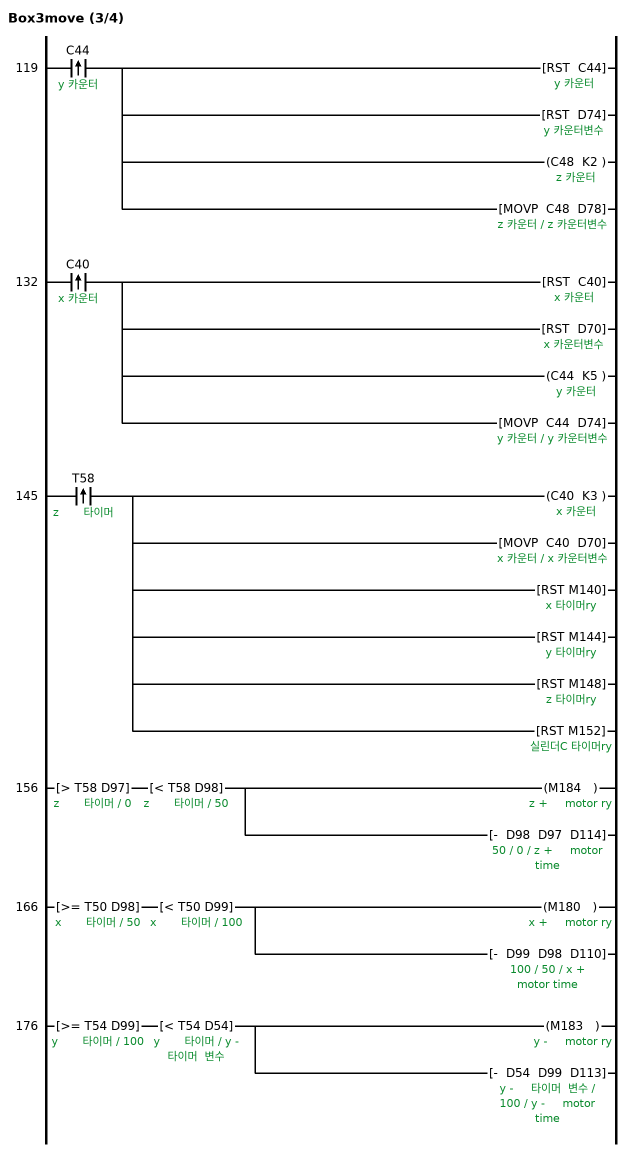
[picture p24: ladder of Box3move, rungs at steps 119 to 176]
119   LDP     C44  ; y 카운터
      RST     C44  ; y 카운터
      RST     D74  ; y 카운터변수
      OUT     C48 K2  ; z 카운터
      MOVP    C48 D78
132   LDP     C40  ; x 카운터
      RST     C40  ; x 카운터
      RST     D70  ; x 카운터변수
      OUT     C44 K5  ; y 카운터
      MOVP    C44 D74
145   LDP     T58  ; z       타이머
      OUT     C40 K3  ; x 카운터
      MOVP    C40 D70
      RST     M140  ; x 타이머ry
      RST     M144  ; y 타이머ry
      RST     M148  ; z 타이머ry
      RST     M152  ; 실린더C 타이머ry
156   LD>     T58 D97  ; z       타이머 / 0
      AND<    T58 D98  ; z       타이머 / 50
      OUT     M184  ; z +     motor ry
      -       D98 D97 D114  ; z +     motor time
166   LD>=    T50 D98  ; x       타이머 / 50
      AND<    T50 D99  ; x       타이머 / 100
      OUT     M180  ; x +     motor ry
      -       D99 D98 D110  ; x +     motor time
176   LD>=    T54 D99  ; y       타이머 / 100
      AND<    T54 D54  ; y       타이머 / y -     타이머  변수
      OUT     M183  ; y -     motor ry
      -       D54 D99 D113  ; y -     motor time
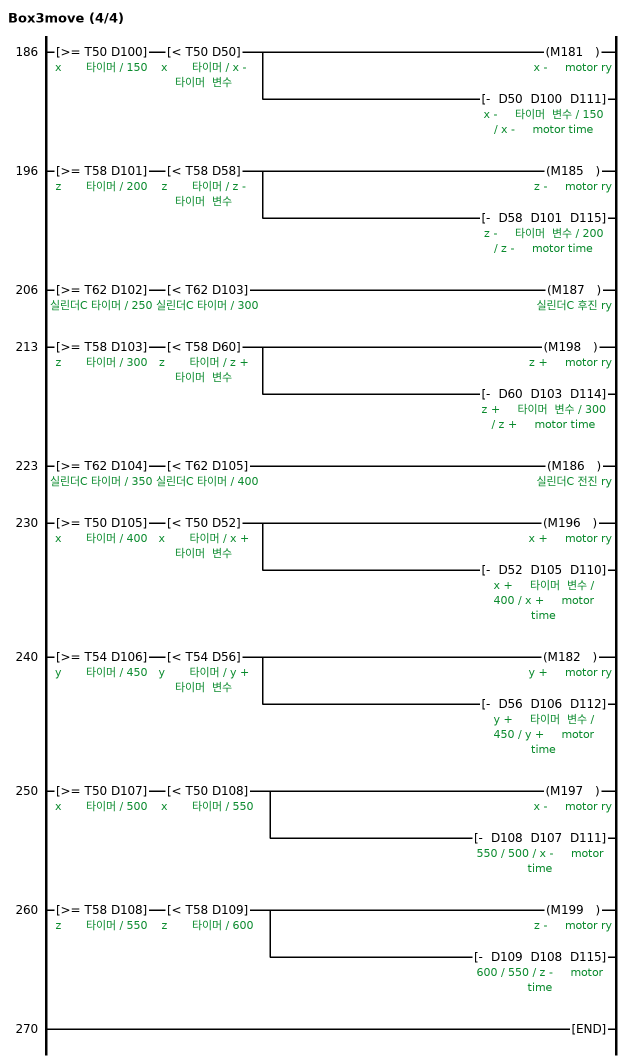
186   LD>=    T50 D100  ; x       타이머 / 150
      AND<    T50 D50  ; x       타이머 / x -     타이머  변수
      OUT     M181  ; x -     motor ry
      -       D50 D100 D111  ; x -     motor time
196   LD>=    T58 D101  ; z       타이머 / 200
      AND<    T58 D58  ; z       타이머 / z -     타이머  변수
      OUT     M185  ; z -     motor ry
      -       D58 D101 D115  ; z -     motor time
206   LD>=    T62 D102  ; 실린더C 타이머 / 250
      AND<    T62 D103  ; 실린더C 타이머 / 300
      OUT     M187  ; 실린더C 후진 ry
213   LD>=    T58 D103  ; z       타이머 / 300
      AND<    T58 D60  ; z       타이머 / z +     타이머  변수
      OUT     M198  ; z +     motor ry
      -       D60 D103 D114
223   LD>=    T62 D104  ; 실린더C 타이머 / 350
      AND<    T62 D105  ; 실린더C 타이머 / 400
      OUT     M186  ; 실린더C 전진 ry
230   LD>=    T50 D105  ; x       타이머 / 400
      AND<    T50 D52  ; x       타이머 / x +     타이머  변수
      OUT     M196  ; x +     motor ry
      -       D52 D105 D110
240   LD>=    T54 D106  ; y       타이머 / 450
      AND<    T54 D56  ; y       타이머 / y +     타이머  변수
      OUT     M182  ; y +     motor ry
      -       D56 D106 D112  ; y +     motor time
250   LD>=    T50 D107  ; x       타이머 / 500
      AND<    T50 D108  ; x       타이머 / 550
      OUT     M197  ; x -     motor ry
      -       D108 D107 D111
260   LD>=    T58 D108  ; z       타이머 / 550
      AND<    T58 D109  ; z       타이머 / 600
      OUT     M199  ; z -     motor ry
      -       D109 D108 D115
270   END
END_PROGRAM

PROGRAM OutPut
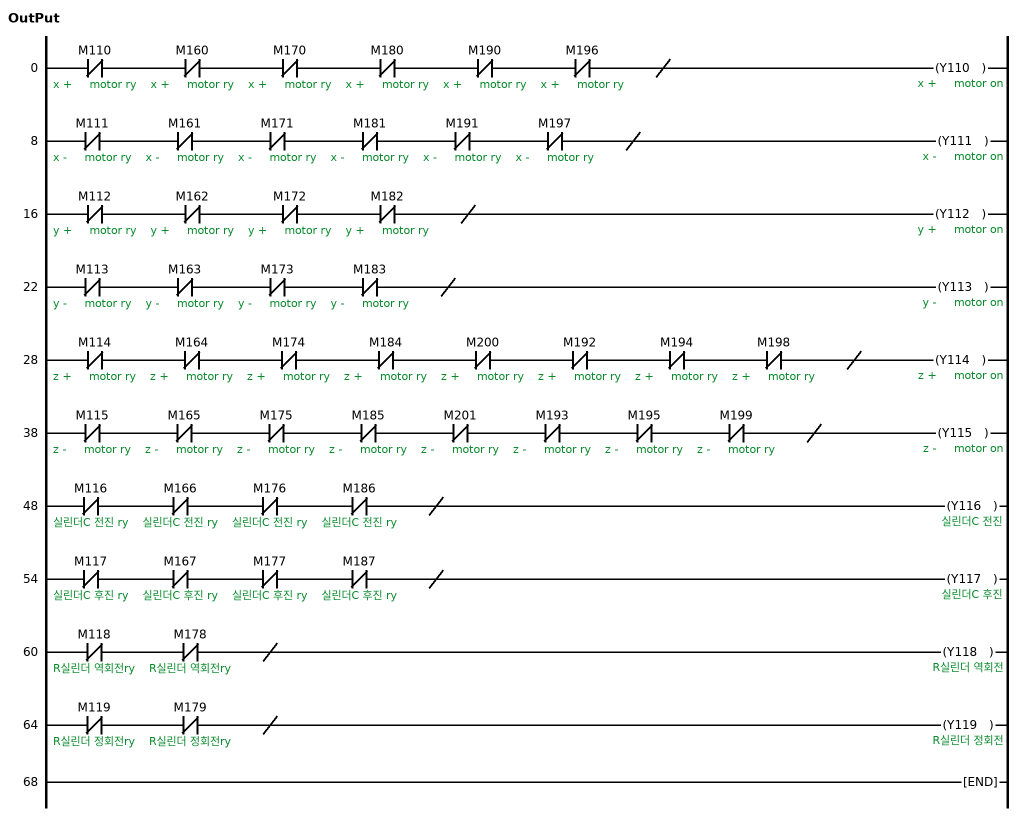
0     LDI     M110  ; x +     motor ry
      ANI     M160  ; x +     motor ry
      ANI     M170  ; x +     motor ry
      ANI     M180  ; x +     motor ry
      ANI     M190  ; x +     motor ry
      ANI     M196  ; x +     motor ry
      INV
      OUT     Y110  ; x +     motor on
8     LDI     M111  ; x -     motor ry
      ANI     M161  ; x -     motor ry
      ANI     M171  ; x -     motor ry
      ANI     M181  ; x -     motor ry
      ANI     M191  ; x -     motor ry
      ANI     M197  ; x -     motor ry
      INV
      OUT     Y111  ; x -     motor on
16    LDI     M112  ; y +     motor ry
      ANI     M162  ; y +     motor ry
      ANI     M172  ; y +     motor ry
      ANI     M182  ; y +     motor ry
      INV
      OUT     Y112  ; y +     motor on
22    LDI     M113  ; y -     motor ry
      ANI     M163  ; y -     motor ry
      ANI     M173  ; y -     motor ry
      ANI     M183  ; y -     motor ry
      INV
      OUT     Y113  ; y -     motor on
28    LDI     M114  ; z +     motor ry
      ANI     M164  ; z +     motor ry
      ANI     M174  ; z +     motor ry
      ANI     M184  ; z +     motor ry
      ANI     M200  ; z +     motor ry
      ANI     M192  ; z +     motor ry
      ANI     M194  ; z +     motor ry
      ANI     M198  ; z +     motor ry
      INV
      OUT     Y114  ; z +     motor on
38    LDI     M115  ; z -     motor ry
      ANI     M165  ; z -     motor ry
      ANI     M175  ; z -     motor ry
      ANI     M185  ; z -     motor ry
      ANI     M201  ; z -     motor ry
      ANI     M193  ; z -     motor ry
      ANI     M195  ; z -     motor ry
      ANI     M199  ; z -     motor ry
      INV
      OUT     Y115  ; z -     motor on
48    LDI     M116  ; 실린더C 전진 ry
      ANI     M166  ; 실린더C 전진 ry
      ANI     M176  ; 실린더C 전진 ry
      ANI     M186  ; 실린더C 전진 ry
      INV
      OUT     Y116  ; 실린더C 전진
54    LDI     M117  ; 실린더C 후진 ry
      ANI     M167  ; 실린더C 후진 ry
      ANI     M177  ; 실린더C 후진 ry
      ANI     M187  ; 실린더C 후진 ry
      INV
      OUT     Y117  ; 실린더C 후진
60    LDI     M118  ; R실린더 역회전ry
      ANI     M178  ; R실린더 역회전ry
      INV
      OUT     Y118  ; R실린더 역회전
64    LDI     M119  ; R실린더 정회전ry
      ANI     M179  ; R실린더 정회전ry
      INV
      OUT     Y119  ; R실린더 정회전
68    END
END_PROGRAM

// device comments not shown above
T4  ; 실린더C 전진    타이머
T5  ; 실린더C 후진    타이머
D22  ; 실린더C 타이머  변수
D24  ; z -     타이머  변수
D62  ; 실린더C 타이머  변수
D64  ; z -     타이머  변수
D116  ; 실린더C 전진 time
D117  ; 실린더C 후진 time
D118  ; R실린더 역회전 time
D119  ; R실린더 정회전 time
